Omron Sysmac Studio project TOF (Sysmac Studio 1.65.0.64007, StandardProject)

# Controller new_Controller_0: NX1P2-1040DT1 version 1.69
Task PrimaryTask (priority 4, period or condition 2000): Program0

VAR_GLOBAL
    BIO_Input_Bit_00 : BOOL;  (* at BuiltInIO://cpu/#0/Input_Bit_00 *)
    BIO_Input_Bit_01 : BOOL;  (* at BuiltInIO://cpu/#0/Input_Bit_01 *)
    BIO_Input_Bit_02 : BOOL;  (* at BuiltInIO://cpu/#0/Input_Bit_02 *)
    BIO_Output_Bit_00 : BOOL;  (* at BuiltInIO://cpu/#0/Output_Bit_00 *)
    BIO_Output_Bit_01 : BOOL;  (* at BuiltInIO://cpu/#0/Output_Bit_01 *)
    IN_StartButton : BOOL;
    IN_Stop_Button : BOOL;
    OUT_Motor1_Start : BOOL;
    OUT_Motor2_Start : BOOL;
    TOF1_ET : TIME;
    TON1_ET : TIME;
END_VAR

PROGRAM Program0
VAR
    Startt : BOOL;
    TOF1 : TOF;
    TON1 : TON;
    TOF11 : TOF;
END_VAR
VAR_EXTERNAL
    BIO_Input_Bit_00 : BOOL;
    IN_StartButton : BOOL;
    BIO_Input_Bit_01 : BOOL;
    IN_Stop_Button : BOOL;
    BIO_Input_Bit_02 : BOOL;
    OUT_Motor1_Start : BOOL;
    BIO_Output_Bit_00 : BOOL;
    OUT_Motor2_Start : BOOL;
    BIO_Output_Bit_01 : BOOL;
    TOF1_ET : TIME;
    TON1_ET : TIME;
END_VAR

(* Section InOut: ladder, written here as Structured Text *)

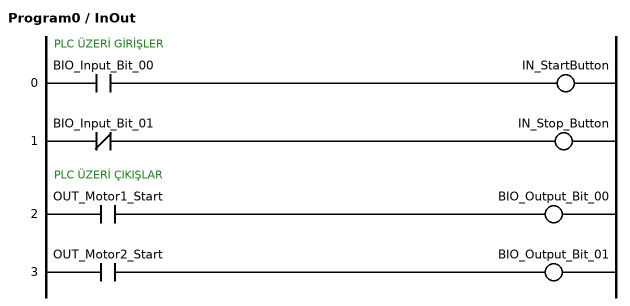
(* Rung 0: PLC ÜZERİ GİRİŞLER *)
IN_StartButton := BIO_Input_Bit_00;
(* Rung 1 *)
IN_Stop_Button := NOT BIO_Input_Bit_01;
(* Rung 2: PLC ÜZERİ ÇIKIŞLAR *)
BIO_Output_Bit_00 := OUT_Motor1_Start;
(* Rung 3 *)
BIO_Output_Bit_01 := OUT_Motor2_Start;

(* Section TONTOF: ladder, written here as Structured Text *)

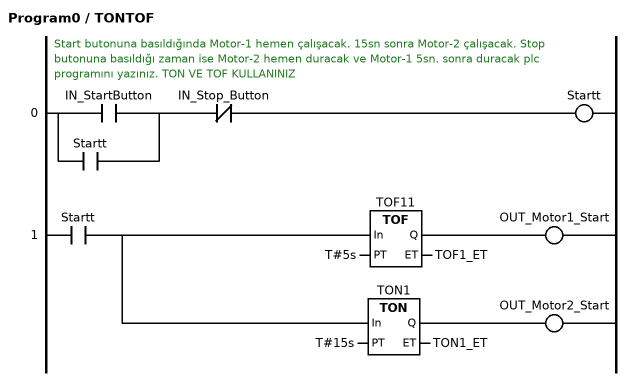
(* Rung 0: Start butonuna basıldığında Motor-1 hemen çalışacak. 15sn sonra Motor-2 çalışacak. Stop butonuna basıldığı zaman ise Motor-2 hemen duracak ve Motor-1 5sn. sonra duracak plc programını yazınız. TON VE TOF KULLANINIZ *)
Startt := (IN_StartButton OR Startt) AND NOT IN_Stop_Button;
(* Rung 1 *)
TOF11(In := Startt, PT := T#5s, ET => TOF1_ET);
OUT_Motor1_Start := TOF11.Q;
TON1(In := Startt, PT := T#15s, ET => TON1_ET);
OUT_Motor2_Start := TON1.Q;
END_PROGRAM